PROGRAM MAIN
VAR
	fbSortingSystemTSM			: FB_SortingSystem_TSM;
END_VAR

// TSMs
	fbSortingSystemTSM();

END_PROGRAM

(* stored: Version 1.1.0.1, ProductVersion 3.1.4024.6
   POU MAIN: Id {d5fa594b-018f-4229-88ac-cd2d1c3a059f}, SpecialFunc None *)
